TYPE ST_Batch :
STRUCT
	sBatchNumber		:STRING;
	sBatchName			:STRING;
	sRecipeName			:STRING;
	sRecipeType			:STRING;
	sProductName		:STRING;
	sComment			:STRING;
	sUser				:STRING;
	sStarted			:STRING;
	sFinished			:STRING;
END_STRUCT
END_TYPE

(* stored: Version 1.1.0.1
   DUT ST_Batch: Id {09c12afd-3bc8-4810-b79e-928305e5884a} *)
